Staubli VAL3: interpolatePos.pgx

program interpolatePos(pointRx x_pStart (dimensions=1), pointRx x_pEnd (dimensions=1))
  local num l_nI
begin
  l_nI=0
  do
    pGoBack[l_nI*10].trsf=interpolateL(x_pStart.trsf,x_pEnd.trsf,l_nI)
    movel(pGoBack[l_nI*10],tTool,mNomSpeed)
    l_nI=l_nI+0.1
  until l_nI>1.05
  waitEndMove()
end
